Staubli VAL3: sCenterTitle.pgx

public program sCenterTitle(string& x_sTitle)
  local num l_nIndex_i
  local string l_sLeadingSpa
  local string l_sTrailingSpa
begin


  //max length 36 characters
  call sCenterString(x_sTitle,asc("=",0),36)


end
